# EPICS autosave request: iocs/scanPBIOC/iocBoot/iocScanPB/auto_settings.req
file "ADScanSim_settings.req",  P=$(P),  R=cam1:
file "NDStdArrays_settings.req",  P=$(P),  R=image1:
file "commonPlugin_settings.req", P=$(P)
